// TIA Portal V20 export
DATA_BLOCK "BK26"   // DB260
// stored: MemoryReserve 100
   VAR
      "X10-1.JR WINDER B-AXIS HOME SENSOR" : Bool := TRUE;
      "X11-1.JR WINDER CLAMP TOP REAR UP/DOWN" : Bool := FALSE;
      "X12-1.MAIN VALVE DIGITAL PRESSURE SWITCH OUT1" : Bool := FALSE;
      "X13-1.JR WINDER CLAMP TOP FRONT UP/DOWN" : Bool := FALSE;
      "X14-1.SPARE" : Bool := FALSE;
      "X15-1.JR WINDER CLAMP TOP REAR PRESSURE SWITCH" : Bool := FALSE;
      "X16-1.SPARE" : Bool := FALSE;
      "X17-1.SPARE" : Bool := FALSE;
      "X10-2.SPARE" : Bool := FALSE;
      "X11-2.SPARE" : Bool := FALSE;
      "X12-2.MAIN VALVE DIGITAL PRESSURE SWITCH OUT2" : Bool := FALSE;
      "X13-2.SPARE" : Bool := FALSE;
      "X14-2.SPARE" : Bool := FALSE;
      "X15-2.JR WINDER CLAMP TOP FRONT PRESSURE SWITCH" : Bool := FALSE;
      "X16-2.SPARE" : Bool := FALSE;
      "X17-2.SPARE" : Bool := FALSE;
   END_VAR
BEGIN
END_DATA_BLOCK
